(* CODESYS project Aventics.library
   Company: Ziga Javornik
   DefaultNamespace: ZigaLibs.Aventics
   Version: 0.0.1.1
   Placeholder: ZigaLibs.Aventics
   Author: Ziga Javornik
   Description: Aventics devices library colelction.
   Title: ZigaLibs.Aventics

Project tree, tasks and I/O mapping:
  libraries: Tc2_Math, * (Beckhoff Automation GmbH); Tc2_Standard, * (Beckhoff Automation GmbH); Tc2_System, * (Beckhoff Automation GmbH); Tc3_Module, * (Beckhoff Automation GmbH); TcUnit, 1.3.1 (www.tcunit.org); ZigaLibs.Core, 0.0.3.7 (Ziga Javornik); ZigaLibs.Logging, 0.0.4.1 (Ziga Javornik)
  DUTs/
  GVLs/
  SOURCE/
    ValveSystem/
      Diagnostics/
        function block FB_XV03_DiagnosticsParser [ST]: OpenLoadCoils, PerformanceDiagnosis
        data type ST_DiagnosticsOptions
        data type ST_XV03_PerformanceDiagnostics
        program XV03_DiagnosticsHelper [ST]: Parse
      Valve/
        data type ST_XV03_CoilInfoData
        data type ST_XV03_ValveInfoData
      function block FB_XV03_ValveSystem [ST]: FB_init, DiagnosticsOptions, Enable, ExecuteDiagnostics, Valves
      data type ST_ValveCoils
      data type T_XV03_ValveSystem
  TESTS/
    Test suites/
      function block FB_XV03_DiagnosisParser_Tests [ST]
      function block FB_XV03ValveSystem_Tests [ST]: Test01_Disabled_AllOutputsAreAlwaysFalse, Test02_Enabled_ExpectCorrectByteBitsSetToTrue
    program PRG_TESTS [ST]
  VISUs/
*)

// SOURCE/ValveSystem/Diagnostics/ST_DiagnosticsOptions
TYPE ST_DiagnosticsOptions :
STRUCT
	Enable	: BOOL;
	Period	: TIME;
END_STRUCT
END_TYPE

// SOURCE/ValveSystem/Diagnostics/ST_XV03_PerformanceDiagnostics
TYPE ST_XV03_PerformanceDiagnostics :
STRUCT
	LOGIC_VOLTAGE_INCORRECT 	: BOOL;
	ACTUATOR_VOLTAGE_OVERRANGE	: BOOL;
	OPEN_LOAD_AT_VALVE_COIL		: BOOL;
	SHORT_CIRCUIT_AT_VALVE_COIL	: BOOL;
	HARDWARE_ERROR				: BOOL;
END_STRUCT
END_TYPE

// SOURCE/ValveSystem/Valve/ST_XV03_CoilInfoData
TYPE ST_XV03_CoilInfoData :
STRUCT
	OpenLoad		: BOOL;
	ShortCircuit	: BOOL;
	Active			: BOOL;
END_STRUCT
END_TYPE

// SOURCE/ValveSystem/Valve/ST_XV03_ValveInfoData
TYPE ST_XV03_ValveInfoData :
STRUCT
	Coil_14	: ST_XV03_CoilInfoData;
	Coil_12	: ST_XV03_CoilInfoData;
END_STRUCT
END_TYPE

// SOURCE/ValveSystem/ST_ValveCoils
TYPE ST_ValveCoils :
STRUCT
	Coils_01_To_08	: BYTE;
	Coils_09_To_16	: BYTE;
	Coils_17_To_24	: BYTE;
	Coils_25_To_32	: BYTE;
	Coils_33_To_40	: BYTE;
	Coils_41_To_48	: BYTE;
END_STRUCT
END_TYPE

// SOURCE/ValveSystem/T_XV03_ValveSystem
TYPE T_XV03_ValveSystem : 
	ARRAY[1..24] OF ST_XV03_ValveInfoData; 
END_TYPE

// SOURCE/ValveSystem/Diagnostics/FB_XV03_DiagnosticsParser
FUNCTION_BLOCK FB_XV03_DiagnosticsParser
VAR_INPUT
END_VAR
VAR_OUTPUT
END_VAR
VAR
END_VAR

METHOD OpenLoadCoils : ARRAY[1..8] OF BOOL
VAR_INPUT
	coils	: USINT;
END_VAR
VAR
	
END_VAR
OpenLoadCoils[1] := coils.0;
OpenLoadCoils[2] := coils.1;
OpenLoadCoils[3] := coils.2;
OpenLoadCoils[4] := coils.3;
OpenLoadCoils[5] := coils.4;
OpenLoadCoils[6] := coils.5;
OpenLoadCoils[7] := coils.6;
OpenLoadCoils[8] := coils.7;
END_METHOD

METHOD PerformanceDiagnosis : REFERENCE TO ST_XV03_PerformanceDiagnostics;
VAR_INPUT
	Value	: USINT;
END_VAR
VAR_INST
	stPerformanceDiagnosis	: ST_XV03_PerformanceDiagnostics;
END_VAR
VAR
	ptr2ndByte	: POINTER TO BYTE;
END_VAR
// 2nd byte is performance diagnosis.
ptr2ndByte := ADR(Value) + SIZEOF(BYTE);
stPerformanceDiagnosis.LOGIC_VOLTAGE_INCORRECT := ptr2ndByte^.0;
stPerformanceDiagnosis.ACTUATOR_VOLTAGE_OVERRANGE := ptr2ndByte^.1;
stPerformanceDiagnosis.OPEN_LOAD_AT_VALVE_COIL := ptr2ndByte^.2;
stPerformanceDiagnosis.SHORT_CIRCUIT_AT_VALVE_COIL := ptr2ndByte^.3;
stPerformanceDiagnosis.HARDWARE_ERROR := ptr2ndByte^.4;
END_METHOD

END_FUNCTION_BLOCK

// SOURCE/ValveSystem/Diagnostics/XV03_DiagnosticsHelper
PROGRAM XV03_DiagnosticsHelper
VAR
END_VAR

METHOD Parse : REFERENCE TO FB_XV03_DiagnosticsParser

VAR_INST
	fbXV03DiagnosisOptions	: FB_XV03_DiagnosticsParser;
END_VAR
Parse REF= fbXV03DiagnosisOptions;
END_METHOD

END_PROGRAM

// SOURCE/ValveSystem/FB_XV03_ValveSystem
FUNCTION_BLOCK FB_XV03_ValveSystem EXTENDS ZigaLibs_Core.FB_HasAmsAddressFromProcessImage
VAR
	_enable					: BOOL;
	_valves					: T_XV03_ValveSystem;
	_logger					: REFERENCE TO ZigaLibs_Logging.I_Logger;
	_diagnosticsOptios		: ST_DiagnosticsOptions;
	_diagnosticsTimer		: Tc2_Standard.TON;
	_init					: BOOL;
END_VAR

VAR
	Coils	AT %Q*			: ST_ValveCoils;
END_VAR

VAR CONSTANT
	MINIMUM_DIAGNOSTICS_PERIOD : TIME := T#1S;
END_VAR

IF NOT _enable THEN
	Coils.Coils_01_To_08 := 0;
	Coils.Coils_09_To_16 := 0;
	Coils.Coils_17_To_24 := 0;
	Coils.Coils_25_To_32 := 0;
	Coils.Coils_41_To_48 := 0;
ELSE
	Coils.Coils_01_To_08.0 := _valves[1].Coil_14.Active;
	Coils.Coils_01_To_08.1 := _valves[1].Coil_12.Active;
	Coils.Coils_01_To_08.2 := _valves[2].Coil_14.Active;
	Coils.Coils_01_To_08.3 := _valves[2].Coil_12.Active;
	Coils.Coils_01_To_08.4 := _valves[3].Coil_14.Active;
	Coils.Coils_01_To_08.5 := _valves[3].Coil_12.Active;
	Coils.Coils_01_To_08.6 := _valves[4].Coil_14.Active;
	Coils.Coils_01_To_08.7 := _valves[4].Coil_12.Active;
	Coils.Coils_09_To_16.0 := _valves[5].Coil_14.Active;
	Coils.Coils_09_To_16.1 := _valves[5].Coil_12.Active;
	Coils.Coils_09_To_16.2 := _valves[6].Coil_14.Active;
	Coils.Coils_09_To_16.3 := _valves[6].Coil_12.Active;
	Coils.Coils_09_To_16.4 := _valves[7].Coil_14.Active;
	Coils.Coils_09_To_16.5 := _valves[7].Coil_12.Active;
	Coils.Coils_09_To_16.6 := _valves[8].Coil_14.Active;
	Coils.Coils_09_To_16.7 := _valves[8].Coil_12.Active;
	
	Coils.Coils_17_To_24.0 := _valves[9].Coil_14.Active;
	Coils.Coils_17_To_24.1 := _valves[9].Coil_12.Active;
	Coils.Coils_17_To_24.2 := _valves[10].Coil_14.Active;
	Coils.Coils_17_To_24.3 := _valves[10].Coil_12.Active;
	Coils.Coils_17_To_24.4 := _valves[11].Coil_14.Active;
	Coils.Coils_17_To_24.5 := _valves[11].Coil_12.Active;
	Coils.Coils_17_To_24.6 := _valves[12].Coil_14.Active;
	Coils.Coils_17_To_24.7 := _valves[12].Coil_12.Active;
	
	Coils.Coils_25_To_32.0 := _valves[13].Coil_14.Active; 
	Coils.Coils_25_To_32.1 := _valves[13].Coil_12.Active; 
	Coils.Coils_25_To_32.2 := _valves[14].Coil_14.Active;
	Coils.Coils_25_To_32.3 := _valves[14].Coil_12.Active;
	Coils.Coils_25_To_32.4 := _valves[15].Coil_14.Active;
	Coils.Coils_25_To_32.5 := _valves[15].Coil_12.Active;
	Coils.Coils_25_To_32.6 := _valves[16].Coil_14.Active;
	Coils.Coils_25_To_32.7 := _valves[16].Coil_12.Active;
	                          
	Coils.Coils_33_To_40.0 := _valves[17].Coil_14.Active;
	Coils.Coils_33_To_40.1 := _valves[17].Coil_12.Active;
	Coils.Coils_33_To_40.2 := _valves[18].Coil_14.Active;
	Coils.Coils_33_To_40.3 := _valves[18].Coil_12.Active;
	Coils.Coils_33_To_40.4 := _valves[19].Coil_14.Active;
	Coils.Coils_33_To_40.5 := _valves[19].Coil_12.Active;
	Coils.Coils_33_To_40.6 := _valves[20].Coil_14.Active;
	Coils.Coils_33_To_40.7 := _valves[20].Coil_12.Active;
	
	Coils.Coils_41_To_48.0 := _valves[21].Coil_14.Active; 
	Coils.Coils_41_To_48.1 := _valves[21].Coil_12.Active; 
	Coils.Coils_41_To_48.2 := _valves[22].Coil_14.Active;
	Coils.Coils_41_To_48.3 := _valves[22].Coil_12.Active;
	Coils.Coils_41_To_48.4 := _valves[23].Coil_14.Active;
	Coils.Coils_41_To_48.5 := _valves[23].Coil_12.Active;
	Coils.Coils_41_To_48.6 := _valves[24].Coil_14.Active;
	Coils.Coils_41_To_48.7 := _valves[24].Coil_12.Active;
END_IF


{warning 'To-do - implement diagnostisc via CoE!'}
_diagnosticsTimer(IN := _diagnosticsOptios.Enable, PT := MAX(_diagnosticsOptios.Period, MINIMUM_DIAGNOSTICS_PERIOD));
IF _diagnosticsTimer.Q OR (NOT _init AND _diagnosticsOptios.Enable) THEN
	ExecuteDiagnostics();
END_IF

IF _diagnosticsOptios.Enable = FALSE THEN
	_init := TRUE;
END_IF

METHOD FB_init : BOOL
VAR_INPUT
	bInitRetains : BOOL; // if TRUE, the retain variables are initialized (warm start / cold start)
	bInCopyCode : BOOL;  // if TRUE, the instance afterwards gets moved into the copy code (online change)
	logger		: REFERENCE TO ZigaLibs_Logging.I_Logger;	// If logging will be used, provide it here. Else set this to 0, internal checks will ommit logging.
END_VAR
IF __ISVALIDREF(logger) THEN
	_logger REF= logger;
END_IF
END_METHOD

{attribute 'monitoring':='call'}
// Gets or sets diagnostics options
PROPERTY DiagnosticsOptions : REFERENCE TO ST_DiagnosticsOptions
GET
DiagnosticsOptions ref= _diagnosticsOptios;
END_GET
END_PROPERTY

{attribute 'monitoring':='call'}
PROPERTY Enable : BOOL
GET
Enable := _enable;
END_GET
SET
_enable := Enable;
END_SET
END_PROPERTY

METHOD PRIVATE ExecuteDiagnostics : BOOL
VAR_INPUT
END_VAR

VAR_INST
	fbCoeReadWrite	: ZigaLibs_Core.FB_CoeReadWrite;
END_VAR
// TO-DO IMPLEMENT!
(*
	fbCoeReadWrite.ReadAny(
		SlaveAddr := THIS^.Ams,
		);
	...
*)

_init := TRUE;
_diagnosticsTimer(IN := FALSE);
END_METHOD

{attribute 'monitoring':='call'}
PROPERTY Valves : REFERENCE TO T_XV03_ValveSystem
GET
Valves REF= _valves;
END_GET
END_PROPERTY

END_FUNCTION_BLOCK

// TESTS/Test suites/FB_XV03_DiagnosisParser_Tests
FUNCTION_BLOCK FB_XV03_DiagnosisParser_Tests EXTENDS FB_TestSuite
VAR_INPUT
END_VAR
VAR_OUTPUT
END_VAR
VAR
	_parser	: FB_XV03_DiagnosticsParser;
END_VAR

END_FUNCTION_BLOCK

// TESTS/Test suites/FB_XV03ValveSystem_Tests
// Subject under test
FUNCTION_BLOCK INTERNAL FB_XV03ValveSystem_Tests EXTENDS FB_TestSuite

// Create instance variables that will be accesible for all tests
VAR

END_VAR

// Call your test methods here
Test01_Disabled_AllOutputsAreAlwaysFalse();
Test02_Enabled_ExpectCorrectByteBitsSetToTrue();

METHOD PRIVATE Test01_Disabled_AllOutputsAreAlwaysFalse

(* Instanced variables are VERY useful for writing tests since tests are run in paralel (by default).
By instantiating local variables that are not placed on the same stack as method (values are retained between calls)
you make sure that the SUT is not changed by some other test. *)
VAR_INST
	emptyArray	: ARRAY[0..SIZEOF(ST_ValveCoils)] OF BYTE;
	fbValves	: FB_XV03_ValveSystem(0);
END_VAR

VAR_INST

END_VAR
// The name of the test, is the same as method name!
IF TcUnit.TEST_ORDERED('Test01_Disabled_AllOutputsAreAlwaysFalse') THEN
	fbValves.Enable := FALSE;
	
	AssertTrue(
		Condition := Tc2_System.MEMCMP(pBuf1 := ADR(emptyArray), pBuf2 := ADR(fbValves.Coils), n := SIZEOF(ST_ValveCoils))  = ZigaLibs_Core.E_MemCmpResults.IDENTICAL,
		Message := 'When disabled, output coils should all be set to 0.');
		
	fbValves.Valves[1].Coil_12.Active := TRUE;
	fbValves.Valves[5].Coil_14.Active := TRUE;
	fbValves.Valves[8].Coil_12.Active := TRUE;
	fbValves.Valves[12].Coil_12.Active := TRUE;
	
	AssertTrue(
		Condition := Tc2_System.MEMCMP(
			pBuf1 := ADR(emptyArray), 
			pBuf2 := ADR(fbValves.Coils), 
			n := SIZEOF(ST_ValveCoils)) = ZigaLibs_Core.E_MemCmpResults.IDENTICAL,
		Message := 'When disabled, output coils should all be set to 0.');

	TcUnit.TEST_FINISHED();	
END_IF
END_METHOD

METHOD PRIVATE Test02_Enabled_ExpectCorrectByteBitsSetToTrue

(* Instanced variables are VERY useful for writing tests since tests are run in paralel (by default).
By instantiating local variables that are not placed on the same stack as method (values are retained between calls)
you make sure that the SUT is not changed by some other test. *)
VAR_INST
		fbValveSystem_XV03	: FB_XV03_ValveSystem(0);
END_VAR

VAR
	iteration						: UINT;
	ptrUsint						: POINTER TO USINT;
	indexValueToAdd					: UINT;
	indexValueToSubstract			: UINT;
	expectedValue					: USINT;
	stringBuilder					: ZigaLibs_Core.FB_StringBuilder;
	addressToAdd					: DWORD;
END_VAR

VAR CONSTANT
	VALVES_PER_BYTE	: REAL := 4.0;
END_VAR
// The name of the test, is the same as method name!
IF TcUnit.TEST_ORDERED('Test02_Enabled_ExpectCorrectByteBitsSetToTrue') THEN
	fbValveSystem_XV03.Enable := TRUE;
	
	FOR iteration := 1 TO 24 BY 1 DO
		// Coil 1 of valve
		fbValveSystem_XV03.Valves[iteration].Coil_14.Active := TRUE;
		fbValveSystem_XV03();
		// add + 1 address when next byte should be looked at (4 valves with 2 coils per byte, 8 bits)
		addressToAdd := LREAL_TO_DWORD((Tc2_Math.FLOOR(TO_LREAL(iteration - 1)/VALVES_PER_BYTE)));
		ptrUsint := ADR(fbValveSystem_XV03.Coils) + addressToAdd;
		expectedValue := LREAL_TO_USINT(EXPT(2, iteration - 1 + indexValueToAdd - indexValueToSubstract));
		AssertTrue(
			Condition := ptrUsint^ = expectedValue,
			Message := stringBuilder.Reset()
				.AddString('Valve ')
				.AddWithDblQuotationMarks(TO_STRING(iteration))
				.AddString(', coil 14 was not opened.')
				.Create());
		
		fbValveSystem_XV03.Valves[iteration].Coil_14.Active := FALSE;
		fbValveSystem_XV03();
		AssertTrue(
			Condition := ptrUsint^ = 0,
			Message := stringBuilder.Reset()
				.AddString('Valve ')
				.AddWithDblQuotationMarks(TO_STRING(iteration))
				.AddString(', coil 14 was not closed.')
				.Create());
		
		// Coil 2 of valve	
		fbValveSystem_XV03.Valves[iteration].Coil_12.Active := TRUE;
		fbValveSystem_XV03();
		// Every 4th valve proceeds to next byte (2 coils per valve, 2x4 = 8 bits = 1 byte, 48 coils total)
		addressToAdd := LREAL_TO_DWORD((Tc2_Math.FLOOR(TO_LREAL(iteration - 1)/VALVES_PER_BYTE)));
		ptrUsint := ADR(fbValveSystem_XV03.Coils) + addressToAdd;
		expectedValue := LREAL_TO_USINT(EXPT(2, iteration + indexValueToAdd - indexValueToSubstract));
		AssertTrue(ptrUsint^ = expectedValue,
			stringBuilder.Reset()
				.AddString('Valve ')
				.AddWithDblQuotationMarks(TO_STRING(iteration))
				.AddString(', coil 12 was not opened.')
				.Create());
				
		indexValueToAdd := indexValueToAdd + 1;
		
		fbValveSystem_XV03.Valves[iteration].Coil_12.Active := FALSE;
		fbValveSystem_XV03();
		AssertTrue(
			Condition := ptrUsint^ = 0,
			Message := stringBuilder.Reset()
				.AddString('Valve ')
				.AddWithDblQuotationMarks(TO_STRING(iteration))
				.AddString(', coil 12 was not closed.')
				.Create());
				
		// In order to have 1 single loop, every loop iteration we need to add 1 value, to increase the 2^n+1 result.
		// When the byte is finished, next iteration would start at 2^n, for example 2^5. But we need to reset back at 1st position.
		// For that reson the substract index will be taken into account in the power calculation and every 4th iteration, 
		// aka 1 byte, the power will be: 2^(iteration - 4*(byte number 0...3) + current coil index (0..1))		
		IF indexValueToAdd = TO_UINT(VALVES_PER_BYTE) THEN
			indexValueToAdd := 0;
			indexValueToSubstract := indexValueToSubstract + TO_UINT(VALVES_PER_BYTE);
		END_IF
	END_FOR
	
	TcUnit.TEST_FINISHED();
END_IF
END_METHOD

END_FUNCTION_BLOCK

// TESTS/PRG_TESTS
PROGRAM INTERNAL PRG_TESTS

(* Instantiate test suites here. Naming convention for tests should be a suffix with _Tests.
Good practice for creating test methods is to end them with _test as well. *)
VAR

	XV03ValveSystem_Tests		: FB_XV03ValveSystem_Tests;
	XV03DiagnosisParser_Tests	: FB_XV03_DiagnosticsParser;
END_VAR

// Run tests in paralel
// TcUnit.RUN();

// Run tests in sequence, one after the other. Uncomment if required.
TcUnit.RUN_IN_SEQUENCE();

END_PROGRAM
